ORGANIZATION_BLOCK "OB 121 Programmierf-OB"	// OB 121
TITLE = Programmierfehler-OB
//Erstellung:
//Datum        Bearbeiter                                                 Version
//--------------------------------------------------------------------------------
//03.06.98     Rainer Schaffert (sra)                                     01.00.00
//
//Änderungen:
//Nr. Datum    Bearb Beschreibung                                   Marke Version
//--------------------------------------------------------------------------------
//01  
//
//________________________________________________________________________________
//OB wird aufgerufen wenn ein Fehler während der Programmbearbeitung auftritt
AUTHOR : sra
FAMILY : AZO
VERSION : 0.0
VAR_TEMP
  OB121_EV_CLASS : BYTE ;	//16#25, Event class 2, Entering event state, Internal fault event
  OB121_SW_FLT : BYTE ;	//16#XX Software programming fault
  OB121_PRIORITY : BYTE ;	//X = Priority of OB where fault occured (Priority of 1 is lowest)
  OB121_OB_NUMBR : BYTE ;	//121 (Organization block 121, OB121)
  OB121_BLK_TYPE : BYTE ;	//16#88/8A/8B/8C/8E Type of block fault occured in
  OB121_RESERVED_1 : BYTE ;	//Reserved for system
  OB121_FLT_REG : WORD ;	//16#XX Specific register that caused fault
  OB121_BLK_NUM : WORD ;	//Number of block that programming fault occured in
  OB121_PRG_ADDR : WORD ;	//Address in block where programming fault occured
  OB121_DATE_TIME : DATE_AND_TIME ;	//Date and time OB121 started
END_VAR
BEGIN
NETWORK
TITLE = Fehlermeldung erzeugen
//Fehlermeldung erzeugen
//
//Fehlercode B#16#21 : BCD-Konvertierungsfehler
//                                
//           B#16#22 : Bereichslängenfehler bei lesen
//
//           B#16#23 : Bereichslängenfehler bei schreiben
//
//           B#16#28 : lesender Zugriff auf ein Byte, Wort oder Doppelwort mit 
//                     einem Pointer, dessen Bitadresse ungleich 0 ist.
//
//           B#16#29 : schreibender Zugriff auf ein Byte, Wort oder Doppelwort 
//                     mit einem Pointer, dessen Bitadresse ungleich 0 ist.
//
//           B#16#24 : Bereichsfehler bei lesen
//
//           B#16#25 : Bereichsfehler bei schreiben
//
//           B#16#26 : Fehler bei Timernummer
//
//           B#16#27 : Fehler bei Zählernummer
//
//           B#16#30 : Schreibender Zugriff auf einen schreibgeschützten Global-DB
//
//           B#16#31 : Schreibender Zugriff auf einen schreibgeschützten 
//                     Instanz-DB
//
//           B#16#32 : DB-Nummernfehler beim Zugriff auf einen Global-DB
//
//           B#16#33 : DB-Nummernfehler beim Zugriff auf einen Instanz-DB
//
//
//
//Fehlermeldung erzeugen
//
//Fehlercode B#16#21 : BCD-Konvertierungsfehler
//                                
//           B#16#22 : Bereichslängenfehler bei lesen
//
//           B#16#23 : Bereichslängenfehler bei schreiben
//
//           B#16#28 : lesender Zugriff auf ein Byte, Wort oder Doppelwort mit 
//                     einem Pointer, dessen Bitadresse ungleich 0 ist.
//
//           B#16#29 : schreibender Zugriff auf ein Byte, Wort oder Doppelwort 
//mit 
//                     einem Pointer, dessen Bitadresse ungleich 0 ist.
//
//           B#16#24 : Bereichsfehler bei lesen
//
//           B#16#25 : Bereichsfehler bei schreiben
//
//           B#16#26 : Fehler bei Timernummer
//
//           B#16#27 : Fehler bei Zählernummer
//
//           B#16#30 : Schreibender Zugriff auf einen schreibgeschützten Global-DB
//
//           B#16#31 : Schreibender Zugriff auf einen schreibgeschützten 
//                     Instanz-DB
//
//           B#16#32 : DB-Nummernfehler beim Zugriff auf einen Global-DB
//
//           B#16#33 : DB-Nummernfehler beim Zugriff auf einen Instanz-DB
//
//           B#16#34 : FC-Nummernfehler beim FC-Aufruf
//
//           B#16#35 : FB-Nummernfehler beim FB-Aufruf
//
//           B#16#3A : Zugriff auf einen nicht geladenen DB
//
//           B#16#3C : Zugriff auf einen nicht geladenen FC
//
//           B#16#3D : Zugriff auf einen nicht geladenen SFC
//
//           B#16#3E : Zugriff auf einen nicht geladenen FB
//
//           B#16#3F : Zugriff auf einen nicht geladenen SFB
//
//
      A(;
      L     #OB121_SW_FLT;
      L     B#16#0;
      <>I;
      );
      =     "DB3 global Info".Fehler_OB_Info.Programmierfehler_OB121;
      L     #OB121_SW_FLT;
      T     "DB3 global Info".Fehler_OB_Info.OB_121_Fault_ID;
END_ORGANIZATION_BLOCK

ORGANIZATION_BLOCK "OB 122 Peripheriezugr-OB"	// OB 122
TITLE = Peripheriezugriffsfehler-OB
//Erstellung:
//Datum        Bearbeiter                                                 Version
//--------------------------------------------------------------------------------
//03.06.98     Rainer Schaffert (sra)                                     01.00.00
//
//Änderungen:
//Nr. Datum    Bearb Beschreibung                                   Marke Version
//--------------------------------------------------------------------------------
//01  
//
//________________________________________________________________________________
//Der OB wird aufgerufen wenn beim Zugreifen auf Daten einer Baugruppe ein Fehler 
//auftritt
AUTHOR : sra
FAMILY : AZO
VERSION : 0.0
VAR_TEMP
  OB122_EV_CLASS : BYTE ;	//16#29, Event class 2, Entering event state, Internal fault event
  OB122_SW_FLT : BYTE ;	//16#XX Software error code
  OB122_PRIORITY : BYTE ;	//X = Priority of OB where fault occured (Priority of 1 is lowest)
  OB122_OB_NUMBR : BYTE ;	//122 (Organization block 122, OB122)
  OB122_BLK_TYPE : BYTE ;	//16#88/8A/8C/8E Type of block fault occured in
  OB122_MEM_AREA : BYTE ;	//Memory area where access error occured
  OB122_MEM_ADDR : WORD ;	//Memory address where access error occured
  OB122_BLK_NUM : WORD ;	//Block number in which error occured
  OB122_PRG_ADDR : WORD ;	//Program address where error occured
  OB122_DATE_TIME : DATE_AND_TIME ;	//Date and time OB1 started
END_VAR
BEGIN
NETWORK
TITLE = Fehlermeldung erzeugen
//Fehlermeldung erzeugen
//
//Fehlercode B#16#42 : Bei S7-300: Periperiezugriffsfehler, lesend
//                     Bei S7-400: Fehler beim ersten Lesezugriff nach auftreten 
//                                 eines Fehlers
//                                
//           B#16#43 : Bei S7-300: Periperiezugriffsfehler, schreibend
//                     Bei S7-400: Fehler beim ersten Schreibzugriff nach         
//                                 auftreten eines Fehlers
//                     
//           B#16#44 : Bei S7-400: Fehler beim n-ten Lesezugriff nach             
//                                 auftreten eines Fehlers
// 
//           B#16#45 : Bei S7-400: Fehler beim n-ten Schreibzugriff nach          
//                                 auftreten eines Fehlers
//
      A(;
      L     #OB122_SW_FLT;
      L     B#16#0;
      <>I;
      );
      =     "DB3 global Info".Fehler_OB_Info.Periphzugriff_OB122;
      L     #OB122_SW_FLT;
      T     "DB3 global Info".Fehler_OB_Info.OB_122_Fault_ID;
END_ORGANIZATION_BLOCK
